(* IEC 61131-3 sources: programs/VI-54/VI-54_20171205/VI-54_20171205/Stations/Screen/LseClass170718/Class/Const, 1 file *)

(* ---- Const.st ---- *)
(*!
<Class
	Name               = "Const"
	Revision           = "1.0"
	RealtimeTask       = "false"
	CyclicTask         = "false"
	BackgroundTask     = "false"
	Sigmatek           = "true"
	OSInterface        = "false"
	HighPriority       = "false"
	Automatic          = "false"
	UpdateMode         = "Prescan"
	IconPath           = ".\Class\Const\Const.ICO"
	SharedCommandTable = "true"
	Objectsize         = "(284,120)"
	Comment            = "constant data, 4 byte">
	<Channels>
		<Server Name="Data" Visualized="true" Initialize="true" WriteProtected="false" Retentive="false" Comment="global interface"/>
	</Channels>
	<Dependencies>
		<Files>
			<File Path=".\Class\Ram\Ram.h" Include="false"/>
		</Files>
	</Dependencies>
</Class>
*)
Const : CLASS
  //Servers:
	Data 	: SvrChCmd_DINT;
  //Clients:
  //Variables:
  //Functions:
  //Tables:
	FUNCTION @STD
		VAR_OUTPUT
			ret_code	: CONFSTATES;
		END_VAR;
	FUNCTION GLOBAL TAB @CT_;
END_CLASS;
